TYPE TcoUrRobotics_O2T_Reg2_IO : 
STRUCT
    bArray AT %Q* : ARRAY[0..99] OF BYTE;
END_STRUCT
END_TYPE

(* stored: Version 1.1.0.1, ProductVersion 3.1.4024.12
   DUT TcoUrRobotics_O2T_Reg2_IO: Id {4039ef47-64e9-0898-2b0d-c0bea1fd783e} *)
